FUNCTION Convert_BYTE_TO_DATE : Hresult
VAR_INPUT
	in : BYTE;
	out : REFERENCE TO DATE;
END_VAR
VAR
	converted : DATE;
END_VAR

converted := BYTE_TO_DATE(in);

IF (DATE_TO_BYTE(converted) <> in) THEN
	Convert_BYTE_TO_DATE := INCOMPATIBLE;
	RETURN;
END_IF

out := converted;

END_FUNCTION

(* stored: Version 1.1.0.1, ProductVersion 3.1.4024.12
   POU Convert_BYTE_TO_DATE: Id {4e9ace99-4eac-4fe5-96e6-5b88e0997ff7}, SpecialFunc None *)
